FUNCTION_BLOCK FB_Read_Only_String_Builder_Adapter IMPLEMENTS I_Read_Only_String_Builder_Adapter
VAR_INPUT
	ipString_Builder : I_String_Builder;
END_VAR

(* Number of bytes allocated in memory for the string builder's contents.*)
PROPERTY _Capacity : T_Size
GET
IF THIS^.ipString_Builder = 0 THEN RETURN; END_IF
_Capacity := THIS^.ipString_Builder._Capacity;
END_GET
END_PROPERTY

(* Current size of string builder contents*)
PROPERTY _Length : T_Size
GET
IF THIS^.ipString_Builder = 0 THEN RETURN; END_IF
_Length := THIS^.ipString_Builder._Length;
END_GET
END_PROPERTY

(* Copies a subset of characters in the string builder from specified position at specified length to a string*)
METHOD Copy_Substring_To : I_Read_Only_String_Builder_Adapter
VAR_INPUT
	Position, Length : T_Size;
	Value : ANY;
END_VAR
Copy_Substring_To := THIS^;
IF THIS^.ipString_Builder = 0 THEN RETURN; END_IF
THIS^.ipString_Builder.Copy_Substring_To(Position, Length, Value);
END_METHOD

(* Copies contents of string builder to given string of any size*)
METHOD Copy_To : I_Read_Only_String_Builder_Adapter
VAR_INPUT
	Value : ANY;
END_VAR
Copy_To := THIS^;
IF THIS^.ipString_Builder = 0 THEN RETURN; END_IF
THIS^.ipString_Builder.Copy_To(Value);
END_METHOD

(* !!!UNSAFE!!! DON'T FORGET TO RELEASE/DELETE FROM	MEMORY WHEN DONE!
 | Get a copy of the internal string buffer at the size of the string length + 1.*)
METHOD Get_Buffer : I_Read_Only_String_Builder_Adapter
VAR_IN_OUT
	pBuffer	: POINTER TO BYTE;
END_VAR
Get_Buffer := THIS^;
IF THIS^.ipString_Builder = 0 THEN RETURN; END_IF
THIS^.ipString_Builder.Get_Buffer(pBuffer);
END_METHOD

(* Retrieves the number of bytes allocated in memory for the string builder's contents.*)
METHOD Get_Capacity : I_Read_Only_String_Builder_Adapter
VAR_OUTPUT
	Capacity	: T_Size;
END_VAR
Get_Capacity := THIS^;
Capacity := THIS^._Capacity;
END_METHOD

(* Gets character at specified position in the string builder*)
METHOD Get_Char : T_Char
VAR_INPUT
	Position	: T_Size;
END_VAR
IF THIS^.ipString_Builder = 0 THEN RETURN; END_IF
Get_Char := THIS^.ipString_Builder.Get_Char(Position);
END_METHOD

(* Retrieves the current size of string builder contents*)
METHOD Get_Length : I_Read_Only_String_Builder_Adapter
VAR_OUTPUT
	Length	: T_Size;
END_VAR
Get_Length := THIS^;
Length := THIS^._Length;
END_METHOD

(* Converts contents of string builder to string and returns them*)
METHOD Get_String : T_Long_String
IF THIS^.ipString_Builder = 0 THEN RETURN; END_IF
Get_String := THIS^.ipString_Builder.Get_String();
END_METHOD

(* Get a subset of characters in the string builder from specified position at specified length and returns them as a string*)
METHOD Get_Substring : T_Long_String
VAR_INPUT
	Position	: T_Size;
	Length	: T_Size;
END_VAR
IF THIS^.ipString_Builder = 0 THEN RETURN; END_IF
Get_Substring := THIS^.ipString_Builder.Get_Substring(Position, Length);
END_METHOD

(* Finds the position of the first instance of a given string in the content's of the string builder from a starting position*)
METHOD Search : I_Read_Only_String_Builder_Adapter
VAR_INPUT
	sValue	: T_Long_String;
	Start_Position	: T_Size;
END_VAR
VAR_OUTPUT
	Position	: T_Size;
END_VAR
Search := THIS^;
IF THIS^.ipString_Builder = 0 THEN RETURN; END_IF
THIS^.ipString_Builder.Search(sValue, Start_Position, Position => Position);
END_METHOD

(* Finds the position of the first instance of a given value in the content's of the string builder from a starting position*)
METHOD Search_Any : I_Read_Only_String_Builder_Adapter
VAR_INPUT
	Value : ANY;
	Start_Position : T_Size;
END_VAR
VAR_OUTPUT
	Position : T_Size := -1;
END_VAR
Search_Any := THIS^;
IF THIS^.ipString_Builder = 0 THEN RETURN; END_IF
THIS^.ipString_Builder.Search_Any(Value, Start_Position, Position => Position);
END_METHOD

(* Appends selected characters from the current string builder to the selected string builder*)
METHOD Split : I_Read_Only_String_Builder_Adapter
VAR_INPUT
	Position : T_Size;
	Length : T_Size;
	ipString_Builder : I_String_Builder;
END_VAR
Split := THIS^;
IF THIS^.ipString_Builder = 0 THEN RETURN; END_IF
THIS^.ipString_Builder.Split(Position, Length, ipString_Builder);
END_METHOD

END_FUNCTION_BLOCK

(* stored: Version 1.1.0.1, ProductVersion 3.1.4024.4
   POU FB_Read_Only_String_Builder_Adapter: Id {5b2f76d6-71b2-41fd-9735-b5916830d938}, SpecialFunc None
   Property _Capacity: Id {5e804c55-c620-4d22-a532-fbaedf7e33f3}
   Get Get: Id {a02353a6-8f43-4024-b756-1b601822b353}
   Property _Length: Id {47428ebe-0553-4546-9fa2-3c3da99dd0e5}
   Get Get: Id {f03399eb-acc0-45e6-b564-02633cd162e1}
   Method Copy_Substring_To: Id {e52e47a2-b7cb-4fc2-937d-d79a7dd6f1c1}
   Method Copy_To: Id {cd0ca31a-3a35-4a56-9e9a-84c2c0a452e5}
   Method Get_Buffer: Id {0e58de1f-9791-406a-84d4-e5bae5496810}
   Method Get_Capacity: Id {e0b2a79e-d112-46c1-a77e-9c5f7b9fc05b}
   Method Get_Char: Id {1af0a8ac-26b2-40b7-8c19-3ef6ce240260}
   Method Get_Length: Id {84f2c33b-4773-4941-aceb-9877e5a12da1}
   Method Get_String: Id {65690ebe-27e3-45fa-ab0e-48130b75ef40}
   Method Get_Substring: Id {9fa3ecbe-5e9c-4351-b490-0efbc9d44201}
   Method Search: Id {cad7533e-4311-4c28-a285-5b01561ebfe0}
   Method Search_Any: Id {67b278b9-ea26-4100-9ab4-f6713e4518df}
   Method Split: Id {90821461-a891-4b50-8400-5b7b505302ad} *)
